(* CODESYS project BagFeedMotorIMove.xml

Project tree, tasks and I/O mapping:
  function block BagFeedMotorIMove [SFC]
*)

// BagFeedMotorIMove
FUNCTION_BLOCK BagFeedMotorIMove
//  .					.					.
VAR_INPUT
	SFCInit: 			BOOL;
	Trigger: 			BOOL;
	Direction: 			UINT; // 1 = Forward, 0 = Reverse;
	Steps: 				UDINT;
	Speed: 				UINT;
	Count: 				UDINT;
	Stop: 				BOOL;
	LabelSensor: 		BOOL;
END_VAR
VAR_OUTPUT
	Forward: 			BOOL;
	Reverse: 			BOOL;
	Complete: 			BOOL;
	ResetCount: 		BOOL;
END_VAR
VAR
	_Direction: 		UINT;
	_Steps: 			UDINT;
	_Speed: 			UINT;
	_Destination:	 	UDINT;
	_80Percent: 		UDINT;
	_Correction: 		UDINT;
	_PID: 				PID;
	
	CTU_0: 				CTU;
	R_TRIG_0: 			R_TRIG;
	F_TRIG_0: 			F_TRIG;
	SensorTrigger: 		BOOL;
	TriggerCounts: 		WORD;
	_EdgeTracker: 		EdgeTracker;
END_VAR

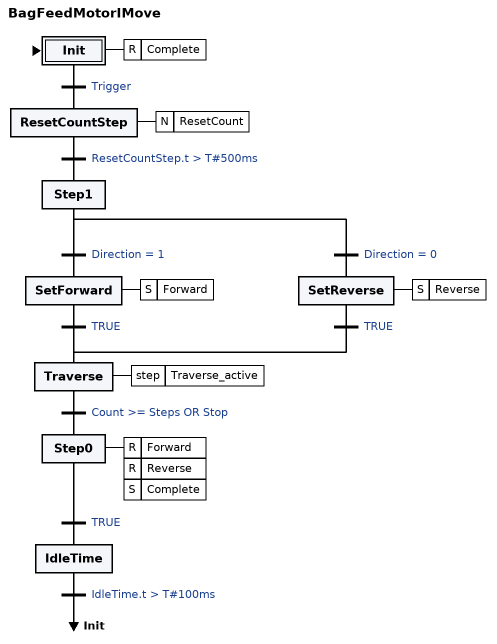
INITIAL_STEP Init:
    Complete(R);
END_STEP
TRANSITION FROM Init TO ResetCountStep
    := Trigger;
END_TRANSITION
STEP ResetCountStep:
    ResetCount(N);
END_STEP
TRANSITION FROM ResetCountStep TO Step1
    := ResetCountStep.t > T#500ms;
END_TRANSITION
STEP Step1:
END_STEP
TRANSITION FROM Step1 TO SetForward
    := Direction = 1;
END_TRANSITION
STEP SetForward:
    Forward(S);
END_STEP
TRANSITION FROM SetForward TO Traverse
    := TRUE;
END_TRANSITION
TRANSITION FROM Step1 TO SetReverse
    := Direction = 0;
END_TRANSITION
STEP SetReverse:
    Reverse(S);
END_STEP
TRANSITION FROM SetReverse TO Traverse
    := TRUE;
END_TRANSITION
STEP Traverse:
    Traverse_active(N);  // step action
END_STEP
TRANSITION FROM Traverse TO Step0
    := Count >= Steps OR Stop;
END_TRANSITION
STEP Step0:
    Forward(R);
    Reverse(R);
    Complete(S);
END_STEP
TRANSITION FROM Step0 TO IdleTime
    := TRUE;
END_TRANSITION
STEP IdleTime:
END_STEP
TRANSITION FROM IdleTime TO Init
    := IdleTime.t > T#100ms;
END_TRANSITION

END_FUNCTION_BLOCK
